Universal Robots PolyScope program: monica_expt_nov_2025.urp

Program monica_expt_nov_2025 (installation=monica_expt_nov_2025 directory=/programs/usbdisk_0 createdIn=3.1.17195.0 lastSavedIn=5.11.7.1010425 robotSerialNumber=20215300688)
Calibrated DH parameters: a=[-0.000141, -0.212179, -0.212308, 0.000047, -0.000122, 0]; d=[0.152006, 27.788784, -19.084997, -8.572607, 0.08546, 0.092122]; alpha=[1.571495, 0.004328, 0.002348, 1.572419, -1.572075, 0]; deltaTheta=[0, 0.515672, 5.863469, -0.095957, 0.000005, 0]
Robot Program (runOnlyOnce=false)
  'Global variables for telling the robot what to do. One instruction at a time.'
  server_ip := "192.168.42.7"
  opcode := "nothing"
  freedrive := False
  op_argument := "null"
  'Initialise gripper'
  Call connect_to_server
  Loop Forever
    Call check_for_instruction
    Call execute_opcode
SubProgram -> execute_opcode
SubProgram -> check_for_instruction
SubProgram -> connect_to_server
SubProgram connect_to_server (keepSynchronizedWithDisk=false)
  'Connect to the Python server'
  Script: textmsg("Connecting to server.")
  open := socket_open(server_ip,8472)
  Loop While (checkContinuously=false) expression=open≟ False
    open := socket_open(server_ip,8472)
    Wait Sleep waitTime=1
  Script: textmsg("Connected.")
SubProgram check_for_instruction (keepSynchronizedWithDisk=false)
  'This one hammers on the server, and checks for new instructions'
  If freedrive ≟ False
    'Only report not busy, if not in freedrive.'
    Script: socket_send_string("I'm not busy. ")
  opcode := "nothing"
  Loop While (checkContinuously=false) expression=opcode≟("nothing")  or opcode≟""
    Script: socket_send_string("Please tell me what to do. ")
    Script: opcode = socket_read_string()
    'Update TCP on the server when there is nothing else to do.'
    current_tcp := get_actual_tcp_pose()
    current_force := force()
    Script: socket_send_string(current_tcp)
    Script: socket_send_string("f=")
    Script: socket_send_string(current_force)
    Script: socket_send_string("; ")
  'Let the server know that we are on it'
  Script: textmsg("Received opcode is: ", opcode)
SubProgram execute_opcode (keepSynchronizedWithDisk=false)
  'Each function is implemented here'
  Script: socket_send_string("I am busy.")
  'Move tool contact point'
  If ( opcode≟"move_tcp" )  and ( freedrive ≟ False )
    Script: socket_send_string("Please send argument.")
    new_pose_arg := socket_read_ascii_float(6)
    If new_pose_arg[0]≠6
      Script: socket_send_string("Invalid argument received for move_tcp")
      Popup Error (haltProgram=false message=move_tcp received an invalid argument. Check the robot log and the server window for details. inputType=Text)
    move_tcp_pose := p[new_pose_arg[1], new_pose_arg[2], new_pose_arg[3], new_pose_arg[4], new_pose_arg[5], new_pose_arg[6]]
    If is_within_safety_limits(move_tcp_pose)≟ True
      Script: movej(move_tcp_pose)
    Else 
      Script: socket_send_string("This pose is not reachable.")
      Popup Error (haltProgram=false message=The specified pose is not reachable. Check the robot's log and the server window for details, inputType=Text)
    Script: textmsg("move_tcp argument is: ", move_tcp_pose)
    new_pose_arg := socket_read_ascii_float(6)
    Script: socket_send_string("I'm not busy.")
  'Update tool contact point'
  If ( opcode≟"update_tcp" )  and ( freedrive ≟ False )
    Script: socket_send_string("Please send argument.")
    new_tcp_arg := socket_read_ascii_float(6)
    If new_tcp_arg[0]≠6
      Script: socket_send_string("Invalid argument received for update_tcp")
      Popup Error (haltProgram=false message=update_tcp received an invalid argument. Check the robot log and the server window for details. inputType=Text)
    new_tcp := p[new_tcp_arg[1], new_tcp_arg[2], new_tcp_arg[3], new_tcp_arg[4], new_tcp_arg[5], new_tcp_arg[6]]
    Script: set_tcp(new_tcp)
    Script: socket_send_string("I'm not busy.")
  'Enable/disable freedrive'
  If opcode≟"freedrive"
    Script: socket_send_string("Please send argument.")
    Script: freedrive_arg = socket_read_string()
    If (freedrive_arg ≟ "ON")  or (freedrive_arg ≟ "On") or (freedrive_arg ≟ "on")
      Script: freedrive_mode()
      Script: freedrive =  True
      Script: socket_send_string("Freedrive mode enabled.")
      Script: textmsg("Freedrive mode is on.")
    Else 
      Script: end_freedrive_mode()
      Script: freedrive =  False
      Script: socket_send_string("Freedrive mode disabled.")
      Script: textmsg("Freedrive mode is off.")
  'Clean up'
  If ( opcode≟"set_gripper" )  and ( freedrive ≟ False )
    Script: socket_send_string("Please send argument.")
    grip_pos_arg := socket_read_ascii_float(1)
    If grip_pos_arg[0]≠1
      Script: socket_send_string("Invalid argument received for set_gripper")
      Popup Error (haltProgram=false message=set_gripper received an invalid argument. Check the robot log and the server window for details. inputType=Text)
    If grip_pos_arg[1] > 100  or  grip_pos_arg[1] < 0
      Script: socket_send_string("Invalid argument received for set_gripper: Number must be between 0 and 100.")
      Popup Error (haltProgram=false message=set_gripper received an invalid argument. Check the robot log and the server window for details. inputType=Text)
    Script: rq_move_and_wait_norm(grip_pos_arg[1])
    Script: socket_send_string("I'm not busy.")
  If (opcode ≟"move_from_via_to")  and (freedrive ≟ False )
    'the big one!'
    Script: socket_send_string("Please send argument.")
    long_argument := socket_read_ascii_float(19)
    If long_argument[0] ≠ 19
      Script: socket_send_string("Invalid argument received for move_from_to!")
      Popup Error (haltProgram=false message=the length of argument for move_from_to wasn't 19. inputType=Text)
    'This elevation tells the robot how much to hover above.'
    elevation := 0.03
    start_pose := p[long_argument[1], long_argument[2], long_argument[3], long_argument[4], long_argument[5], long_argument[6]]
    start_pose_elev := p[long_argument[1], long_argument[2], long_argument[3] + elevation, long_argument[4], long_argument[5], long_argument[6]]
    via_pose := p[long_argument[7], long_argument[8], long_argument[9], long_argument[10], long_argument[11], long_argument[12]]
    end_pose := p[long_argument[13], long_argument[14], long_argument[15], long_argument[16], long_argument[17], long_argument[18]]
    end_pose_elev := p[long_argument[13], long_argument[14], long_argument[15] + elevation, long_argument[16], long_argument[17], long_argument[18]]
    open_grip_size := long_argument[19]
    Script: socket_send_string("I am busy.")
    'now we are ready to move the robot.'
    Script: rq_move_norm(open_grip_size)
    Script: movej(start_pose_elev)
    Script: movej(start_pose)
    Script: rq_move_and_wait_norm(100)
    Script: movej(start_pose_elev)
    Script: movec(via_pose, end_pose_elev)
    Script: movej(end_pose)
    Script: rq_move_and_wait_norm(open_grip_size)
    Script: movej(end_pose_elev)
    Script: rq_move_norm(open_grip_size)
    Script: rq_move_and_wait_norm(100)
    Script: socket_send_string("I'm not busy.")
  If (opcode≟"move_tcp_rpy") and freedrive ≟  False
    'This is move_tcp, but we convert the RPY vector to robot rotation.'
    Script: socket_send_string("Please send argument.")
    new_pose_arg := socket_read_ascii_float(6)
    If new_pose_arg[0] ≠ 6
      Script: socket_send_string("Invalid argument received for move_tcp")
      Popup Error (haltProgram=false message=move_tcp received an invalid argument. Check the robot log and the server window for details. inputType=Text)
    rpy_vector := [new_pose_arg[4], new_pose_arg[5], new_pose_arg[6]]
    'convert the rpy to rot'
    rot_vector := rpy2rotvec(rpy_vector)
    converted_tcp := p[new_pose_arg[1], new_pose_arg[2], new_pose_arg[3], rot_vector[0], rot_vector[1], rot_vector[2]]
    If is_within_safety_limits(converted_tcp)
      Script: movej(converted_tcp)
    Else 
      Script: socket_send_string("This pose is not reachable.")
      Popup Error (haltProgram=false message=The specified pose is not reachable. Check the robot's log and the server window for details, inputType=Text)
    Script: socket_send_string("I'm not busy.")
  opcode := "nothing"
